// TIA Portal project "ProjectFinal" (V16)

(* hardware
DEVICE "S7-1200 station_1"  S7-1200 Station
   slot 0: "Rack_0"  S7-1200 Rack  Rack  V1.0
   slot 1: "PLC_1"  CPU 1214C AC/DC/Rly  6ES7 214-1BG40-0XB0  V4.2
   slot 2: "DQ 8xRelay_1"  SM 1222 DQ8 x relay  6ES7 222-1HF32-0XB0  V2.0
   slot 3: "DQ 8xRelay_2"  6ES7 222-1HF30-0XB0  V1.0
*)

// ===== PLC "PLC_1"  CPU 1214C AC/DC/Rly =====

VAR_GLOBAL   // PLC tag table "Default tag table"
   "Slider1P2" AT %Q0.0 : Bool;
   "Slider1P1" AT %Q0.1 : Bool;
   "Pinza1O" AT %Q0.2 : Bool;
   "Pinza1C" AT %Q0.3 : Bool;
   "Elevador1U" AT %Q0.4 : Bool;
   "Turn1" AT %Q0.5 : Bool;
   "Slider3P1" AT %Q0.6 : Bool;
   "Slider3P2" AT %Q0.7 : Bool;
   "Pinza2C" AT %Q1.0 : Bool;
   "Turn2" AT %Q1.1 : Bool;
   "CodoP2" AT %Q2.3 : Bool;
   "CodoP1" AT %Q2.4 : Bool;
   "Turn3" AT %Q2.5 : Bool;
   "Elevador3U" AT %Q2.6 : Bool;
   "Pinza3O" AT %Q2.7 : Bool;
   "Pinza3C" AT %Q3.4 : Bool;
   "Slider4P2" AT %Q3.5 : Bool;
   "Pinza4C" AT %Q3.6 : Bool;
   "Slider4P1" AT %Q3.7 : Bool;
   "Slider4.2P2" AT %Q2.0 : Bool;
   "Slider4.2P1" AT %Q2.1 : Bool;
   "Elevador4U" AT %Q2.2 : Bool;
   "Emergencia" AT %Q3.1 : Bool;
   "Elevador4D" AT %Q3.0 : Bool;
END_VAR

ORGANIZATION_BLOCK "Main"   // OB1, LAD, ProgramCycle
TITLE = "Main Program Sweep (Cycle)"
{ S7_Optimized_Access := 'TRUE' }
VERSION : 0.1
   VAR_INPUT
      Initial_Call : Bool;   // Initial call of this OB
      Remanence : Bool;   // =True, if remanent data are available
   END_VAR
BEGIN
END_ORGANIZATION_BLOCK